// Mitsubishi GX Works2 project: testPLc   PLC: FX3U/FX3UC

PROGRAM MAIN
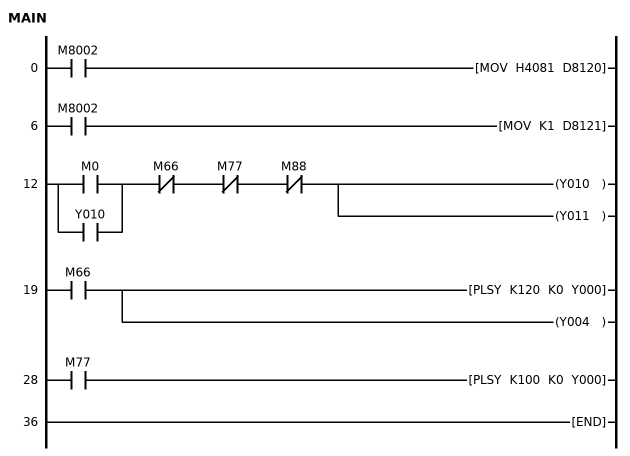
0     LD      M8002
      MOV     H4081 D8120
6     LD      M8002
      MOV     K1 D8121
12    LD      M0
      OR      Y010
      ANI     M66
      ANI     M77
      ANI     M88
      OUT     Y010
      OUT     Y011
19    LD      M66
      PLSY    K120 K0 Y000
      OUT     Y004
28    LD      M77
      PLSY    K100 K0 Y000
36    END
END_PROGRAM
